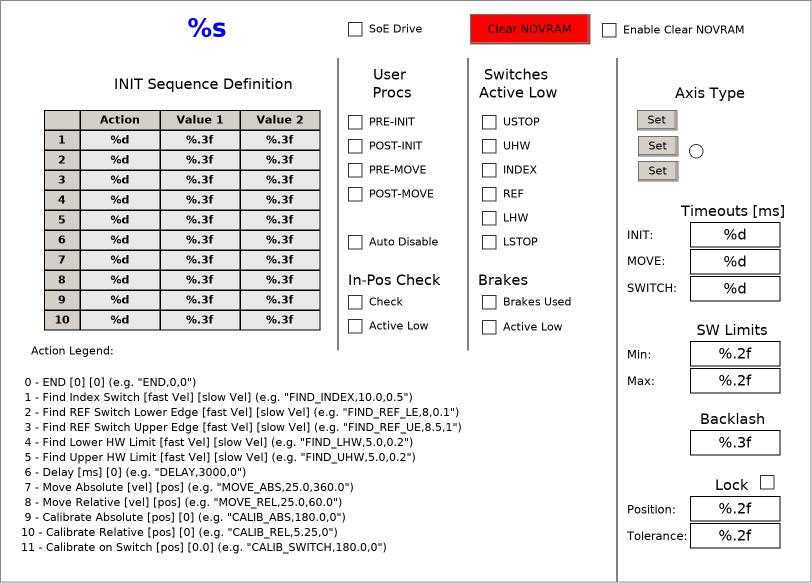
VISUALIZATION GUI_TEMPLATE_MOTOR_CONFIG  // 812x583
VAR_IN_OUT
	m_Instance : FB_MOTOR;
END_VAR
VAR
	bEnableNovramClear:	BOOL := FALSE;
END_VAR
    Label (28,336 150x30), "Action Legend:"
    Label (18,371 600x23), "0 - END [0] [0] (e.g. "END,0,0")"
    Label (18,386 600x23), "1 - Find Index Switch [fast Vel] [slow Vel] (e.g. "FIND_INDEX,10.0,0.5")"
    Label (18,401 600x23), "2 - Find REF Switch Lower Edge [fast Vel] [slow Vel] (e.g. "FIND_REF_LE,8,0.1")"
    Label (18,416 600x23), "3 - Find REF Switch Upper Edge [fast Vel] [slow Vel] (e.g. "FIND_REF_UE,8.5,1")"
    Label (18,431 600x23), "4 - Find Lower HW Limit [fast Vel] [slow Vel] (e.g. "FIND_LHW,5.0,0.2")"
    Label (18,446 600x23), "5 - Find Upper HW Limit [fast Vel] [slow Vel] (e.g. "FIND_UHW,5.0,0.2")"
    Label (18,476 600x23), "7 - Move Absolute [vel] [pos] (e.g. "MOVE_ABS,25.0,360.0")"
    Label (18,491 600x23), "8 - Move Relative [vel] [pos] (e.g. "MOVE_REL,25.0,60.0")"
    Label (18,506 600x23), "9 - Calibrate Absolute [pos] [0] (e.g. "CALIB_ABS,180.0,0")"
    Label (18,521 600x23), "10 - Calibrate Relative [pos] [0] (e.g. "CALIB_REL,5.25,0")"
    Label (18,461 600x23), "6 - Delay [ms] [0] (e.g. "DELAY,3000,0")"
    Label (18,536 600x23), "11 - Calibrate on Switch [pos] [0.0] (e.g. "CALIB_SWITCH,180.0,0")"
    Label (59,69 289x30), "INIT Sequence Definition"
    Label (462,54 113x59), "Switches Active Low"
    Checkbox (480,110 93x24), "USTOP", variable: m_Instance.cfg.bArrActiveLow[5].bValue, invisible if: false, input disabled if: false
    Checkbox (480,134 93x24), "UHW", variable: m_Instance.cfg.bArrActiveLow[4].bValue, invisible if: false, input disabled if: false
    Checkbox (480,158 93x24), "INDEX", variable: m_Instance.cfg.bArrActiveLow[3].bValue, invisible if: false, input disabled if: false
    Checkbox (480,182 93x24), "REF", variable: m_Instance.cfg.bArrActiveLow[2].bValue, invisible if: false, input disabled if: false
    Checkbox (480,206 93x24), "LHW", variable: m_Instance.cfg.bArrActiveLow[1].bValue, invisible if: false, input disabled if: false
    Checkbox (480,230 93x24), "LSTOP", variable: m_Instance.cfg.bArrActiveLow[0].bValue, invisible if: false, input disabled if: false
    Rectangle (87,7 240x42), "%s", text variable: m_Instance.sName
    Label (678,196 132x30), "Timeouts [ms]"
    Label (665,78 90x30), "Axis Type"
    Label (687,315 90x30), "SW Limits"
    Label (475,265 103x30), "Brakes"
    Label (685,404 95x30), "Backlash"
    RadioButton (687,112 114x78), variable: m_Instance.cfg.nAxisType-1, input disabled if: FALSE
        Areas[0]: Text=Linear
        Areas[1]: Text=Circular
        Areas[2]: Text=Circular-Opt
        p3166011961: Cicular-Optimised
    Checkbox (480,290 110x24), "Brakes Used", variable: m_Instance.cfg.bUseBrake, invisible if: false, input disabled if: false
    Checkbox (480,315 105x24), "Active Low", tooltip "Brake Feedback Signal is Active Low", variable: m_Instance.cfg.bActiveLowBrake, invisible if: false, input disabled if: false
    Rectangle (690,430 90x25), "%.3f", tooltip "Positive, negative or zero (no backlash)", text variable: m_Instance.cfg.lrBacklash
        OnMouseDown: write the text variable via Default
    Button (637,110 40x20), "Set"
        OnMouseClick: execute { m_Instance.cfg.nAxisType := 1; }
    Button (638,136 40x20), "Set"
        OnMouseClick: execute { m_Instance.cfg.nAxisType := 2; }
    Button (638,161 40x20), "Set"
        OnMouseClick: execute { m_Instance.cfg.nAxisType := 3; }
    Rectangle (690,341 90x25), "%.2f", tooltip "Setting both limits to 0 means that limits are not used.", text variable: m_Instance.cfg.lrMinPosition
        OnMouseDown: write the text variable via Default
    Rectangle (690,368 90x25), "%.2f", tooltip "Setting both limits to 0 means that limits are not used.", text variable: m_Instance.cfg.lrMaxPosition
        OnMouseDown: write the text variable via Default
    Label (624,340 37x29), "Min:"
    Label (624,366 37x30), "Max:"
    Label (624,220 49x30), "INIT:"
    Label (624,246 49x30), "MOVE:"
    Rectangle (690,222 90x25), "%d", tooltip "INIT sequence timeout in [ms].", text variable: m_Instance.cfg.nTimeoutInit
        OnMouseDown: write the text variable via Default
    Rectangle (690,249 90x25), "%d", tooltip "INIT sequence timeout in [ms].", text variable: m_Instance.cfg.nTimeoutMove
        OnMouseDown: write the text variable via Default
    Line (468,350) (468,58)
    Line (617,581) (617,58)
    Rectangle (690,276 90x25), "%d", tooltip "Switch exit timeout in [ms].", text variable: m_Instance.cfg.nTimeoutSwitch
        OnMouseDown: write the text variable via Default
    Label (624,273 60x30), "SWITCH:"
    Rectangle (80,110 80x20), "Action"
    Rectangle (160,110 80x20), "Value 1"
    Rectangle (240,110 80x20), "Value 2"
    Rectangle (44,130 36x20), "1"
    Rectangle (44,110 36x20)
    Rectangle (80,130 80x20), "%d", text variable: m_Instance.cfg.strArrInitSeq[1].nAction
        OnMouseDown: write the text variable via Default
    Rectangle (160,130 80x20), "%.3f", text variable: m_Instance.cfg.strArrInitSeq[1].lrValue1
        OnMouseDown: write the text variable via Default
    Rectangle (240,130 80x20), "%.3f", text variable: m_Instance.cfg.strArrInitSeq[1].lrValue2
        OnMouseDown: write the text variable via Default
    Rectangle (44,150 36x20), "2"
    Rectangle (80,150 80x20), "%d", text variable: m_Instance.cfg.strArrInitSeq[2].nAction
        OnMouseDown: write the text variable via Default
    Rectangle (160,150 80x20), "%.3f", text variable: m_Instance.cfg.strArrInitSeq[2].lrValue1
        OnMouseDown: write the text variable via Default
    Rectangle (240,150 80x20), "%.3f", text variable: m_Instance.cfg.strArrInitSeq[2].lrValue2
        OnMouseDown: write the text variable via Default
    Rectangle (44,170 36x20), "3"
    Rectangle (80,170 80x20), "%d", text variable: m_Instance.cfg.strArrInitSeq[3].nAction
        OnMouseDown: write the text variable via Default
    Rectangle (160,170 80x20), "%.3f", text variable: m_Instance.cfg.strArrInitSeq[3].lrValue1
        OnMouseDown: write the text variable via Default
    Rectangle (240,170 80x20), "%.3f", text variable: m_Instance.cfg.strArrInitSeq[3].lrValue2
        OnMouseDown: write the text variable via Default
    Rectangle (44,190 36x20), "4"
    Rectangle (80,190 80x20), "%d", text variable: m_Instance.cfg.strArrInitSeq[4].nAction
        OnMouseDown: write the text variable via Default
    Rectangle (160,190 80x20), "%.3f", text variable: m_Instance.cfg.strArrInitSeq[4].lrValue1
        OnMouseDown: write the text variable via Default
    Rectangle (240,190 80x20), "%.3f", text variable: m_Instance.cfg.strArrInitSeq[4].lrValue2
        OnMouseDown: write the text variable via Default
    Rectangle (44,210 36x20), "5"
    Rectangle (80,210 80x20), "%d", text variable: m_Instance.cfg.strArrInitSeq[5].nAction
        OnMouseDown: write the text variable via Default
    Rectangle (160,210 80x20), "%.3f", text variable: m_Instance.cfg.strArrInitSeq[5].lrValue1
        OnMouseDown: write the text variable via Default
    Rectangle (240,210 80x20), "%.3f", text variable: m_Instance.cfg.strArrInitSeq[5].lrValue2
        OnMouseDown: write the text variable via Default
    Rectangle (44,230 36x20), "6"
    Rectangle (80,230 80x20), "%d", text variable: m_Instance.cfg.strArrInitSeq[6].nAction
        OnMouseDown: write the text variable via Default
    Rectangle (160,230 80x20), "%.3f", text variable: m_Instance.cfg.strArrInitSeq[6].lrValue1
        OnMouseDown: write the text variable via Default
    Rectangle (240,230 80x20), "%.3f", text variable: m_Instance.cfg.strArrInitSeq[6].lrValue2
        OnMouseDown: write the text variable via Default
    Rectangle (44,250 36x20), "7"
    Rectangle (80,250 80x20), "%d", text variable: m_Instance.cfg.strArrInitSeq[7].nAction
        OnMouseDown: write the text variable via Default
    Rectangle (160,250 80x20), "%.3f", text variable: m_Instance.cfg.strArrInitSeq[7].lrValue1
        OnMouseDown: write the text variable via Default
    Rectangle (240,250 80x20), "%.3f", text variable: m_Instance.cfg.strArrInitSeq[7].lrValue2
        OnMouseDown: write the text variable via Default
    Rectangle (44,270 36x20), "8"
    Rectangle (80,270 80x20), "%d", text variable: m_Instance.cfg.strArrInitSeq[8].nAction
        OnMouseDown: write the text variable via Default
    Rectangle (160,270 80x20), "%.3f", text variable: m_Instance.cfg.strArrInitSeq[8].lrValue1
        OnMouseDown: write the text variable via Default
    Rectangle (240,270 80x20), "%.3f", text variable: m_Instance.cfg.strArrInitSeq[8].lrValue2
        OnMouseDown: write the text variable via Default
    Rectangle (44,290 36x20), "9"
    Rectangle (80,290 80x20), "%d", text variable: m_Instance.cfg.strArrInitSeq[9].nAction
        OnMouseDown: write the text variable via Default
    Rectangle (160,290 80x20), "%.3f", text variable: m_Instance.cfg.strArrInitSeq[9].lrValue1
        OnMouseDown: write the text variable via Default
    Rectangle (240,290 80x20), "%.3f", text variable: m_Instance.cfg.strArrInitSeq[9].lrValue2
        OnMouseDown: write the text variable via Default
    Rectangle (44,310 36x20), "10"
    Rectangle (80,310 80x20), "%d", text variable: m_Instance.cfg.strArrInitSeq[10].nAction
        OnMouseDown: write the text variable via Default
    Rectangle (160,310 80x20), "%.3f", text variable: m_Instance.cfg.strArrInitSeq[10].lrValue1
        OnMouseDown: write the text variable via Default
    Rectangle (240,310 80x20), "%.3f", text variable: m_Instance.cfg.strArrInitSeq[10].lrValue2
        OnMouseDown: write the text variable via Default
    Line (338,350) (338,58)
    Label (345,54 94x59), "User Procs"
    Checkbox (346,110 106x24), "PRE-INIT", variable: m_Instance.cfg.bExecUserPreInit, invisible if: false, input disabled if: false
    Checkbox (346,134 106x24), "POST-INIT", variable: m_Instance.cfg.bExecUserPostInit, invisible if: false, input disabled if: false
    Checkbox (346,158 106x24), "PRE-MOVE", variable: m_Instance.cfg.bExecUserPreMove, invisible if: false, input disabled if: false
    Checkbox (346,182 106x24), "POST-MOVE", variable: m_Instance.cfg.bExecUserPostMove, invisible if: false, input disabled if: false
    Label (687,470 90x30), "Lock"
    Rectangle (690,496 90x25), "%.2f", tooltip "If the motor is locked, during INIT the motor will not move and its position will be set to this value.", text variable: m_Instance.cfg.lrLockPos
        OnMouseDown: write the text variable via Default
    Rectangle (690,523 90x25), "%.2f", tooltip "The motor will not move, if the target position is closer to the locked position than this value.", text variable: m_Instance.cfg.lrLockTol
        OnMouseDown: write the text variable via Default
    Label (624,495 56x29), "Position:"
    Label (624,521 63x30), "Tolerance:"
    Checkbox (758,470 30x24), tooltip "Flag if motor is locked", variable: m_Instance.cfg.bLock, invisible if: false, input disabled if: false
    Checkbox (346,290 106x24), "Check", tooltip "If active, check if the in-pos signal is active after the move completes. If it is not, it's a failure.", variable: m_Instance.cfg.bCheckInPos, invisible if: false, input disabled if: false
    Checkbox (346,314 107x24), "Active Low", tooltip "If checked, In-Position feedback signal is active low", variable: m_Instance.cfg.bActiveLowInPos, invisible if: false, input disabled if: false
    Checkbox (346,230 127x24), "Auto Disable", tooltip "Auto Disable Motor After Move", variable: m_Instance.cfg.bDisableAfterMove, invisible if: false, input disabled if: false
    Label (345,265 103x30), "In-Pos Check"
    Button (470,14 120x30), "Clear NOVRAM", tooltip "Clear NOVRAM. Use it with care! This is needed ONLY if NOVRAM was previously used for data structures different than T_MOTOR_CFG (or for previous versions of T_MOTOR_CFG). Bring the motor to NOT_READY first and then clear NOVRAM.", input disabled if: bEnableNovramClear=false OR m_Instance.nNOVRAM_DevId=0
        OnMouseUp: execute {
            m_Instance.ctrl.bLocalCmd := TRUE;
            m_Instance.ctrl.nCommand:=E_MOTOR_COMMAND.CLEAR_NOVRAM;
            m_Instance.ctrl.bExecute:=(TRUE);
        }
    Checkbox (600,18 160x24), "Enable Clear NOVRAM", variable: bEnableNovramClear, invisible if: false, input disabled if: false
    Checkbox (346,17 90x24), "SoE Drive", tooltip "Check the box if this is an SoE drive (Sercos over EtherCAT) , e.g. AX5000", variable: m_Instance.cfg.bSoE_Drive, invisible if: false, input disabled if: false
END_VISUALIZATION

(* stored: Version 1.1.0.1, ProductVersion 3.1.4022.16
   Visu GUI_TEMPLATE_MOTOR_CONFIG: Id {bc44775d-30aa-44fb-b24c-1a7b3572e812} *)
